// TIA Portal V18 export
DATA_BLOCK "FDBACK error_n0005-ms1-k3001_SN10-1"   // DB29, F_DB
{ DB_Accessible_From_OPC_UA := 'FALSE' }
// stored: DBAccessibleFromOPCUA false, DBAccessibleFromWebserver false, InstanceOfName 03_FDBACK error, InstanceOfType FB
"03_FDBACK error"
   // VAR_INPUT
   //    Commissioning_bypass : Bool;
   //    "FDBACK ERROR 1" : Bool;
   //    "FDBACK ERROR 2" : Bool;
   //    "FDBACK ERROR 3" : Bool;
   //    "FDBACK ERROR 4" : Bool;
   //    "FDBACK ERROR 5" : Bool;
   //    "FDBACK ERROR 6" : Bool;
   //    "FDBACK ERROR 7" : Bool;
   //    "FDBACK ERROR 8" : Bool;
   // END_VAR
   // VAR_OUTPUT
   //    "Cumulative FDBACK" : Bool;
   //    "ERROR 1" : Bool;
   //    "ERROR 2" : Bool;
   //    "ERROR 3" : Bool;
   //    "ERROR 4" : Bool;
   //    "ERROR 5" : Bool;
   //    "ERROR 6" : Bool;
   //    "ERROR 7" : Bool;
   //    "ERROR 8" : Bool;
   // END_VAR
BEGIN
END_DATA_BLOCK
